FUNCTION_BLOCK OutputDecompressor (* Basic Function Block Type *)
  (* Standard: 61499-2 *)
  (* Version 0.0, 6/21/2018, Rediska, nxtControl GmbH, Template *)
  PACKAGE Main;
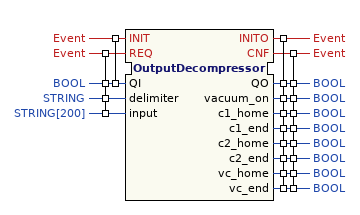
  EVENT_INPUT
    INIT WITH QI; (* Initialization Request *)
    REQ WITH QI, delimiter, input; (* Normal Execution Request *)
  END_EVENT
  EVENT_OUTPUT
    INITO WITH QO, vacuum_on, c1_home, c1_end, c2_home, c2_end, vc_home, vc_end; (* Initialization Confirm *)
    CNF WITH QO, vacuum_on, c1_home, c1_end, c2_home, c2_end, vc_home, vc_end; (* Execution Confirmation *)
  END_EVENT
  VAR_INPUT
    QI : BOOL; (* Input event qualifier *)
    delimiter : STRING;
    input : STRING[200];
  END_VAR
  VAR_OUTPUT
    QO : BOOL; (* Output event qualifier *)
    vacuum_on : BOOL;
    c1_home : BOOL;
    c1_end : BOOL;
    c2_home : BOOL;
    c2_end : BOOL;
    vc_home : BOOL;
    vc_end : BOOL;
  END_VAR
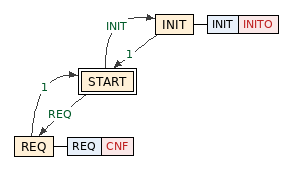
  EC_STATES
    START; (* Initial State *)
    INIT : INIT -> INITO; (* Initialization *)
    REQ : REQ -> CNF; (* Normal execution *)
  END_STATES
  EC_TRANSITIONS
    START TO INIT := INIT;
    INIT TO START := 1;
    START TO REQ := REQ;
    REQ TO START := 1;
  END_TRANSITIONS
  ALGORITHM INIT IN ST: (* Initialization algorithm *)
QO := TRUE;
  END_ALGORITHM
  ALGORITHM REQ IN ST: (* Normally executed algorithm *)
VAR
	length: INT;
	i : INT;
	prev: INT;
	substr : ARRAY[1..7] OF STRING;
	num : INT;
	cur: INT;
END_VAR
length := DINT_TO_INT(LEN(input));
prev := 1;
cur := 1;
FOR i := 1 TO length DO
	IF (MID(input,1,i) = delimiter) THEN
		substr[cur] := MID(input, i - prev, prev);
		cur := cur + 1;
		prev := i + 1;
	END_IF;
END_FOR;
vacuum_on := STRING_TO_BOOL(substr[1]);
c1_home := STRING_TO_BOOL(substr[2]);
c1_end := STRING_TO_BOOL(substr[3]);

c2_home := STRING_TO_BOOL(substr[4]);
c2_end := STRING_TO_BOOL(substr[5]);
vc_home := STRING_TO_BOOL(substr[6]);
vc_end := STRING_TO_BOOL(substr[7]);
  END_ALGORITHM
END_FUNCTION_BLOCK
